PROGRAM MAIN
VAR
END_VAR


// ***********************************************************************************
//
// USI Mendrisio, Largo Bernasconi 2, CH-6850 Mendrisio
// ETH Zurich, Building HIF E26, Laura-Hezner-Weg 7, CH-8093 Zürich
//
// ***********************************************************************************
//
// PROJECT     :  Clay Printing Controller
// FUNCTION    :  Main
// AUTHOR      :  WeiTing Chen
// EMAIL       :  chen@mesh.ch
// Copyright   :  USI FMAA Mendrisio(CH) 2025
//
// ***********************************************************************************


// Control Mode select
P_Control_Mode();

// Operation Mode select
// TODO: Implementation of the operation mode. Now everything services as laptop mode.
IF GVL.b_mode_laptop THEN
	P_Laptop_Operate();
ELSIF GVL.b_mode_robot THEN
	P_Laptop_Operate();
ELSIF GVL.b_mode_manual THEN
	P_Laptop_Operate();
END_IF

END_PROGRAM

(* stored: Version 1.1.0.1, ProductVersion 3.1.4024.15
   POU MAIN: Id {e0e3ca32-8ac9-4c9e-aa5e-a282e7142877}, SpecialFunc None *)
